(* IEC 61131-3 sources: Industry-PLC-LLM/data/PLCBEAD_repo/PLCBEAD_PLCEmbed-main/PLC-BEAD/Source/GEB/UDINT_TO_TIME, 1 file *)

(* ---- UDINT_TO_TIME.ST ---- *)
FUNCTION _UDINT_TO_TIME:TIME

	VAR_INPUT
		IN :	UDINT;
	END_VAR

	_UDINT_TO_TIME := DINT_TO_TIME(UDINT_TO_DINT(IN));

END_FUNCTION

PROGRAM program0
  VAR
	  IN :	UDINT;
    CEIL5_OUT : TIME;
  END_VAR

  CEIL5_OUT := _UDINT_TO_TIME(IN);
END_PROGRAM
